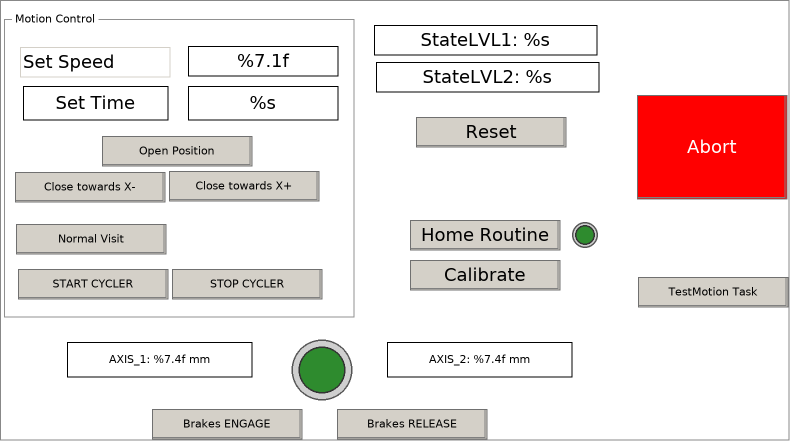
VISUALIZATION TestMotionGUI  // 790x441
    GroupBox (4,11 350x306), "Motion Control"
        Rectangle (19,75 145x34), "Set Time", input disabled if: MAIN.testMotionState<>100;
            OnMouseUp: write GVL.expoTime via Edit, format %7.1f
        Rectangle (184,75 150x34), "%s", text variable: GVL.expoTime
        Button (14,258 150x30), "START CYCLER", input disabled if: MAIN.testMotionState <> 100;
            OnMouseUp: execute { MAIN.testMotionState:=3100; }
    Button (152,409 150x30), "Brakes ENGAGE", input disabled if: MAIN.axis[0].brake=FALSE AND MAIN.axis[1].brake=FALSE;
        OnMouseClick: execute { MAIN.axis[0].brake:=FALSE; MAIN.axis[1].brake:=FALSE; }
    Button (337,409 150x30), "Brakes RELEASE", input disabled if: MAIN.axis[0].brake=TRUE AND MAIN.axis[1].brake=TRUE;
        OnMouseClick: execute { MAIN.axis[0].brake:=TRUE; MAIN.axis[1].brake:=TRUE; }
    Lamp1 (287,335 70x70), variable: MAIN.axis[0].brake and MAIN.axis[1].brake;, style: Lamp-Lamp1-Green
    Rectangle (67,342 185x35), "AXIS_1: %7.4f mm", text variable: MAIN.axis[0].axisRef.NcToPlc.ActPos
    Rectangle (387,342 185x35), "AXIS_2: %7.4f mm", text variable: MAIN.axis[1].axisRef.NcToPlc.ActPos
    Button (638,277 150x30), "TestMotion Task", input disabled if: GVL.task=2;
        OnMouseUp: execute { GVL.task:=2; }
    Button (416,117 150x30), "Reset"
        OnMouseUp: execute { MAIN.reset := TRUE; }
    Button (637,95 150x104), "Abort"
        OnMouseUp: execute { MAIN.abort := TRUE; }
    Rectangle (374,25 223x30), "StateLVL1: %s", text variable: MAIN.testMotionState;
    Button (410,220 150x30), "Home Routine", input disabled if: MAIN.testMotionState <> 100;
        OnMouseUp: execute { MAIN.testMotionState := 400; }
    Button (102,136 150x30), "Open Position", input disabled if: MAIN.testMotionState <> 100;
        OnMouseUp: execute { MAIN.testMotionState:=1000; }
    Textfield (20,47 150x30), "Set Speed", input disabled if: MAIN.testMotionState<>100;
        OnMouseUp: write MAIN.speed via Default, min 0, max 2000, format %7.1f
    Rectangle (188,46 150x30), "%7.1f", text variable: MAIN.speed
    Button (169,171 150x30), "Close towards X+", input disabled if: MAIN.testMotionState <> 100;
        OnMouseUp: execute { MAIN.testMotionState:=1100; }
    Button (15,172 150x30), "Close towards X-", input disabled if: MAIN.testMotionState <> 100;
        OnMouseUp: execute { MAIN.testMotionState:=1200; }
    Button (16,224 150x30), "Normal Visit", input disabled if: MAIN.testMotionState <> 100;
        OnMouseUp: execute { MAIN.testMotionState:=2000; }
    Lamp1 (570,220 30x30), variable: MAIN.axis[0].axisRef.Status.Homed and MAIN.axis[1].axisRef.Status.Homed;, style: Lamp-Lamp1-Green
    Button (410,260 150x30), "Calibrate", input disabled if: MAIN.testMotionState <> 100;
        OnMouseUp: execute { MAIN.testMotionState:=8000; }
    Button (172,269 150x30), "STOP CYCLER"
        OnMouseUp: execute { MAIN.stop:=TRUE; }
    Rectangle (376,62 223x30), "StateLVL2: %s", text variable: MAIN.motion.stateLVL2;
END_VISUALIZATION

(* stored: Version 1.1.0.1, ProductVersion 3.1.4020.12
   Visu TestMotionGUI: Id {623b2af7-4d31-4390-b4d9-d32c32e32a74} *)
